FUNCTION_BLOCK FB_ClockPulse
VAR_INPUT
	bStart:BOOL;
	delOn: TIME:=T#500MS;
	delOff: TIME:= T#200MS;
END_VAR
VAR_OUTPUT
	bExecuteClock: BOOL;
END_VAR
VAR
	fbTimer1, fbTimer2: TON;
END_VAR

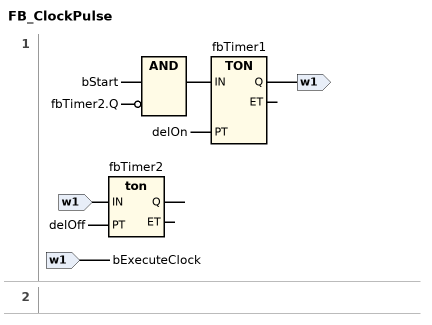
// NETWORK 1
fbTimer1(IN := bStart AND NOT fbTimer2.Q, PT := delOn); // TON
fbTimer2(IN := fbTimer1.Q, PT := delOff); // ton
bExecuteClock := fbTimer1.Q;

// NETWORK 2

END_FUNCTION_BLOCK

(* stored: Version 1.1.0.1, ProductVersion 3.1.4024.12
   POU FB_ClockPulse: Id {fdc97072-5d93-4c6e-a94c-d4c6f179c9b3}, SpecialFunc None *)
